Yaskawa INFORM job: TSYNC-R-TEST.JBI

/JOB
//NAME TSYNC-R-TEST
///FOLDERNAME INNE
//POS
///NPOS 0,0,0,0,0,0
//INST
///DATE 2023/10/04 15:12
///ATTR SC,RW,RJ
////FRAME ROBOT
NOP
*LABEL
MACRO1 MJ#(1) ARGF1
TIMER T=1.00
MACRO1 MJ#(1) ARGF10
TIMER T=1.00
MACRO1 MJ#(1) ARGF100
TIMER T=1.00
MACRO1 MJ#(1) ARGF255
JUMP *LABEL
END
